PROGRAM MAIN
VAR
END_VAR

VAR_INPUT
END_VAR

// Starten der Anlage
Reaktoranlage();
Systemauswertung();

// Starten des Kommunikationsauswertung
Connect();
Disconnect();

// Lesen von RezeptStatusWord
Read();

// Auswertung des RezeptControlWords für Sekundärreaktor
UpdateSek();

// Auswertung des RezeptStatusWords für Systemupdate
UpdateSys();

// Starten des Rezeptes
Rezept_1();

END_PROGRAM

(* stored: Version 1.1.0.1, ProductVersion 3.1.4024.12
   POU MAIN: Id {076a6edd-7aae-4d3b-ac7f-5e66ffd1b567}, SpecialFunc None *)
